//---------------------------------------------------------------------------------------------------------------
//
//  HAUD 2024.03.18
//
//  - XTS_TRANSPORT_LAYER
//
//  fb_TransportUnit
//  - Ctrl/STate interface, reacts to change of command
//    - Cmd(E_TRANSPORT_CTRL)
//
//  - controls members via structures and interfaces for getting XTS in defined state
//    - CMD_INIT:
//        - XPU is initialized:         XTS_CMD_INIT + PROGRESS_DONE
//        - XPU cyclic checks enabled:  XTS_IDLE     + PROGRESS_WORKING
//        - XPU detects mover:          _XpuState.Check == MOVER_ID_DETECTION_VALID
//
//    - CMD_IDLE
//      - Cyclic Checks of XPU and CaGroup
//        - XPU cyclic checks enabled:  XTS_IDLE     + PROGRESS_WORKING
//
//
//  CTRL / STATE --> see proprerties
//  structs for use of function block via mapping
//  cyclic check for new command
//
//  VAR INPUT / OUTPUT --> see properties
//
//---------------------------------------------------------------------------------------------------------------
// This SOFTWARE is provided as an Example by THE PROVIDER "as is" and "with all faults." THE PROVIDER makes no 
// representations or warranties of any kind concerning the safety, suitability, lack of viruses, inaccuracies, 
// typographical errors, or other harmful components of this SOFTWARE. There are inherent dangers in the use of 
// any software, and you are solely responsible for determining whether this SOFTWARE is compatible with your 
// equipment and other software installed on your equipment. You are also solely responsible for the protection 
// of your equipment and backup of your data, and THE PROVIDER will not be liable for any damages you may suffer 
// in connection with using, modifying, or distributing this SOFTWARE.
//---------------------------------------------------------------------------------------------------------------
FUNCTION_BLOCK fb_TransportUnit
VAR
  _eCheck                       : E_XTS_TRANSPORT_CHECK;

  // Transport Ctrl/State
  _stCtrl                       : REFERENCE TO ST_XTS_TRANSPORT_CTRL;
  _stState                      : REFERENCE TO ST_XTS_TRANSPORT_STATE;


  // execute transport commands
  _eCmd,
  _eCmdOld                      : E_XTS_TRANSPORT_CTRL;

  // execution state
  _eState                       : E_XTS_TRANSPORT_STATE;

  // execution result
  _eJobResult,
  _eResult                      : E_PROGRESS;


  // members of transport
  _XpuCtrl                      : REFERENCE TO ST_XPU_CTRL;                     // processing unit ctrl
  _XpuState                     : REFERENCE TO ST_XPU_STATE;                    // processing unit state
  _XpuInfo                      : REFERENCE TO ST_XPU_INFO;                     // processing unit information

  _GroupItf                     : I_XtsTransport_CaGroup;                       // group methods
  _GroupInfo                    : REFERENCE TO ST_GROUP_INFO;                   // info from group

  _MoverItf                     : REFERENCE TO ARRAY[1..MAX_MOVER] OF I_XtsTransport_Mover;   // mover methods
  _MoverInfo                    : REFERENCE TO ARRAY[1..MAX_MOVER] OF ST_MOVER_INFO;          // info from mover
  _MoverLastPosition            : REFERENCE TO ARRAY[1..MAX_MOVER] OF LREAL;                  // last commanded position of mover
  _MoverLastGap                 : REFERENCE TO ARRAY[1..MAX_MOVER] OF LREAL;                  // last commanded gapp of mover

  _StationStart                 : REFERENCE TO ST_STATION_PARAMETER;            // position, gap, dynamic constraints for sending all mover to start position

  // stations lists
  _ItfStationList               : REFERENCE TO ARRAY[1..MAX_STATION]  OF I_Station_LinkedList;  // access to all stations lists

  // station controls
  _StationControl               : REFERENCE TO ARRAY[1..MAX_STATION]  OF ST_STATION_CTRL;

  // station states
  _StationState                 : REFERENCE TO ARRAY[1..MAX_STATION]  OF ST_STATION_STATE;


  // access to stations methods by interface
  _ItfStationCtrl               : REFERENCE TO ARRAY[1..MAX_STATION]  OF I_XtsTransport_Station;

  _nStartStation                : UINT;

  _stMoverDataSend              : ST_STATION_MOVER_DATA;    // mover ticket data

  _stListResult                 : ST_STATION_LIST_RESULT;   // Xts station linkedlist entry

  _eMessageLevel                : E_MessageType;
  _stMsg                        : ST_Message;
END_VAR

IF NOT Check() THEN RETURN; END_IF

_stMsg.eDevice                  := XtsTransportUnit + 1;

_eCmd                           := _stCtrl.Cmd;
// check for command change
// get state for cmd
IF (_eCmd <> _eCmdOld)
THEN
  _eState                       := Cmd(_eCmd);
  _eCmdOld                      := _eCmd;

  IF (_eMessageLevel > E_MessageType.eMessageWarning)
  THEN
    _stMsg.eType                := E_MessageType.eMessageInfo;
    _stMsg.eSubdevice           := e_Subdevice.TransportUnit_General;
    _stMsg.iErrorNumber         := 0;
    _stMsg.sText                := concat( 'Command: ', TO_STRING(_eCmd));
    _stMsg.sText                := concat(_stMsg.sText, ': ');
    _stMsg.sText                := concat(_stMsg.sText, TO_STRING(_eResult));
    f_MessageSet(_stMsg);
  END_IF
END_IF

CASE _eResult
OF
  E_PROGRESS.PROGRESS_INVALID:
    _stState.State                := TO_UINT(_eResult);

  E_PROGRESS.PROGRESS_ERROR:
    _stState.State                := _eState + E_PROGRESS.PROGRESS_ERROR;

  E_PROGRESS.PROGRESS_DONE:
    _stState.State                := _eState + E_PROGRESS.PROGRESS_DONE;

    IF (_GroupInfo.GroupErrorStop) OR
       (_GroupInfo.GroupError)     OR
       NOT (_XpuInfo.AllPositionsValid)
    THEN
      _eResult                  := E_PROGRESS.PROGRESS_ERROR;
    END_IF
ELSE
  _stState.State                  := _eState + _eResult;

  CASE _eState
  OF
    E_XTS_TRANSPORT_STATE.TRANSPORT_INIT:
      _eResult                  := XpuInit(TRUE);
  
    E_XTS_TRANSPORT_STATE.TRANSPORT_IDLE:
      _eResult                  := f_GetProgress(_XpuState.State);
  
      IF (_GroupInfo.GroupErrorStop) OR
         (_GroupInfo.GroupError)     OR
         NOT (_XpuInfo.AllPositionsValid)
      THEN
        _eResult                := E_PROGRESS.PROGRESS_ERROR;
      END_IF
  
    E_XTS_TRANSPORT_STATE.TRANSPORT_MOVER_ENABLE:
      _eResult                  := MoverEnableAll(TRUE);
  
    E_XTS_TRANSPORT_STATE.TRANSPORT_MOVER_DISABLE:
      _eResult                  := MoverDisableAll(TRUE);

    E_XTS_TRANSPORT_STATE.TRANSPORT_MOVER_HALT_CA:
      _eResult                  := MoverHaltAll(TRUE);

    E_XTS_TRANSPORT_STATE.TRANSPORT_MOVER_STOP:
      _eResult                  := MoverStopAll(TRUE);
  
    E_XTS_TRANSPORT_STATE.TRANSPORT_GROUP_CLEAR:
      _eResult                  := GroupClear(TRUE);
  
    E_XTS_TRANSPORT_STATE.TRANSPORT_GROUP_BUILD:
      _eResult                  := GroupBuild(TRUE);
  
    E_XTS_TRANSPORT_STATE.TRANSPORT_GROUP_ENABLE:
      _eResult                  := GroupEnable(TRUE);

    E_XTS_TRANSPORT_STATE.TRANSPORT_GROUP_STOP:
      _eResult                  := GroupStop(TRUE);

    E_XTS_TRANSPORT_STATE.TRANSPORT_START:
      _eResult                  := TransportStart(TRUE);
  
    E_XTS_TRANSPORT_STATE.TRANSPORT_RESTART:
      _eResult                  := TransportRestart(TRUE);
  ELSE
    _eResult                    := E_PROGRESS.PROGRESS_INVALID;
  END_CASE

END_CASE

_stState.XpuState                 := _XpuState;
_stState.XpuInfo                  := _XpuInfo;
_stState.GroupInfo                := _GroupInfo;

METHOD PRIVATE Check  : BOOL
VAR_INST
  _idx        : UINT;
END_VAR

IF NOT __ISVALIDREF(_stCtrl)
THEN
  _eCheck                     := E_XTS_TRANSPORT_CHECK.POINTER_NULL_CTRL;
  RETURN;
END_IF

IF NOT __ISVALIDREF(_stState)
THEN
  _eCheck                     := E_XTS_TRANSPORT_CHECK.POINTER_NULL_STATE;
  RETURN;
END_IF

_stState.Check                  := _eCheck;

IF NOT __ISVALIDREF(_XpuCtrl)
THEN
  _eCheck                     := E_XTS_TRANSPORT_CHECK.POINTER_NULL_XPU_CTRL;
  RETURN;
END_IF

IF NOT __ISVALIDREF(_XpuState)
THEN
  _eCheck                     := E_XTS_TRANSPORT_CHECK.POINTER_NULL_XPU_STATE;
  RETURN;
END_IF

IF NOT __ISVALIDREF(_XpuInfo)
THEN
  _eCheck                     := E_XTS_TRANSPORT_CHECK.POINTER_NULL_XPU_INFO;
  RETURN;
END_IF

IF NOT (_GroupItf <> 0)
THEN
  _eCheck                     := E_XTS_TRANSPORT_CHECK.POINTER_NULL_GROUP_ITF;
  RETURN;
END_IF

IF NOT __ISVALIDREF(_GroupInfo)
THEN
  _eCheck                     := E_XTS_TRANSPORT_CHECK.POINTER_NULL_GROUP_INFO;
  RETURN;
END_IF

IF NOT __ISVALIDREF(_MoverItf)
THEN
  _eCheck                     := E_XTS_TRANSPORT_CHECK.POINTER_NULL_MOVER;
  RETURN;
END_IF

FOR _idx := 1 TO MAX_MOVER
DO
  IF NOT (_MoverItf[_idx] <> 0)
  THEN
    _eCheck                   := E_XTS_TRANSPORT_CHECK.POINTER_NULL_MOVER_ITF;
    RETURN;
  END_IF
END_FOR

IF NOT __ISVALIDREF(_MoverInfo)
THEN
  _eCheck                     := E_XTS_TRANSPORT_CHECK.POINTER_NULL_MOVER_INFO;
  RETURN;
END_IF

IF NOT __ISVALIDREF(_MoverLastPosition)
THEN
  _eCheck                     := E_XTS_TRANSPORT_CHECK.POINTER_NULL_MOVER_LAST_POS;
  RETURN;
END_IF

IF NOT __ISVALIDREF(_MoverLastGap)
THEN
  _eCheck                     := E_XTS_TRANSPORT_CHECK.POINTER_NULL_MOVER_LAST_GAP;
  RETURN;
END_IF

IF NOT __ISVALIDREF(_StationStart)
THEN
  _eCheck                     := E_XTS_TRANSPORT_CHECK.POINTER_NULL_STATION_START;
  RETURN;
END_IF

IF NOT __ISVALIDREF(_ItfStationList)
THEN
  _eCheck                     := E_XTS_TRANSPORT_CHECK.POINTER_NULL_STATION_ITF;
  RETURN;
END_IF

IF NOT __ISVALIDREF(_StationControl)
THEN
  _eCheck                     := E_XTS_TRANSPORT_CHECK.POINTER_NULL_STATION_CONTROL;
  RETURN;
END_IF

IF NOT __ISVALIDREF(_StationState)
THEN
  _eCheck                     := E_XTS_TRANSPORT_CHECK.POINTER_NULL_STATION_STATE;
  RETURN;
END_IF

IF NOT __ISVALIDREF(_ItfStationCtrl)
THEN
  _eCheck                     := E_XTS_TRANSPORT_CHECK.POINTER_NULL_STATION_CTRL_ITF;
  RETURN;
END_IF

FOR _idx := 1 TO MAX_STATION
DO
  IF NOT (_ItfStationCtrl[_idx] <> 0)
  THEN
    _eCheck                   := E_XTS_TRANSPORT_CHECK.POINTER_NULL_STATION_CTRL_ITF;
    RETURN;
  END_IF
END_FOR


_eCheck                       := E_XTS_TRANSPORT_CHECK.DONE_CHECK;
Check                         := TRUE;
END_METHOD

METHOD PRIVATE Cmd : E_XTS_TRANSPORT_STATE
VAR_INPUT
  Ctrl      : E_XTS_TRANSPORT_CTRL;
END_VAR
VAR_INST
  _eState   : E_XTS_TRANSPORT_STATE;
END_VAR
IF NOT Check() THEN RETURN; END_IF


CASE Ctrl
OF
  E_XTS_TRANSPORT_CTRL.CMD_NULL:  // clear all method calls
    _eState               := E_XTS_TRANSPORT_STATE.TRANSPORT_NULL;
    _eResult              := XpuInit         (FALSE);
    _eResult              := GroupClear      (FALSE);
    _eResult              := GroupBuild      (FALSE);
    _eResult              := GroupEnable     (FALSE);
    _eResult              := GroupStop       (FALSE);
    _eResult              := MoverEnableAll  (FALSE);
    _eResult              := MoverDisableAll (FALSE);
    _eResult              := MoverHaltAll    (FALSE);
    _eResult              := MoverStopAll    (FALSE);
    _eResult              := TransportStart  (FALSE);
    _eResult              := TransportRestart(FALSE);

  E_XTS_TRANSPORT_CTRL.CMD_INIT:  // clear methods for initialization
    _eState               := E_XTS_TRANSPORT_STATE.TRANSPORT_INIT;
    _eResult              := XpuInit(FALSE);


ELSE
  IF NOT (_XpuState.Init = E_XPU_INIT.INIT_DONE)
  THEN
    // no init, no further commands possible
    _eState               := E_XTS_TRANSPORT_STATE.TRANSPORT_INVALID;
  ELSE
    CASE Ctrl
    OF
      E_XTS_TRANSPORT_CTRL.CMD_IDLE:
        _eState           := E_XTS_TRANSPORT_STATE.TRANSPORT_IDLE;

      E_XTS_TRANSPORT_CTRL.CMD_MOVER_ENABLE:
        _eState           := E_XTS_TRANSPORT_STATE.TRANSPORT_MOVER_ENABLE;
        _eResult          := MoverEnableAll(FALSE);

      E_XTS_TRANSPORT_CTRL.CMD_MOVER_DISABLE:
        _eState           := E_XTS_TRANSPORT_STATE.TRANSPORT_MOVER_DISABLE;
        _eResult          := MoverDisableAll(FALSE);

      E_XTS_TRANSPORT_CTRL.CMD_MOVER_HALT_CA:
        _eState           := E_XTS_TRANSPORT_STATE.TRANSPORT_MOVER_HALT_CA;
        _eResult          := MoverHaltAll(FALSE);

      E_XTS_TRANSPORT_CTRL.CMD_MOVER_STOP:
        _eState           := E_XTS_TRANSPORT_STATE.TRANSPORT_MOVER_STOP;
        _eResult          := MoverStopAll(FALSE);

      E_XTS_TRANSPORT_CTRL.CMD_GROUP_CLEAR:
        _eState           := E_XTS_TRANSPORT_STATE.TRANSPORT_GROUP_CLEAR;
        _eResult          := GroupClear (FALSE);

      E_XTS_TRANSPORT_CTRL.CMD_GROUP_BUILD:
        _eState           := E_XTS_TRANSPORT_STATE.TRANSPORT_GROUP_BUILD;
        _eResult          := GroupBuild (FALSE);

      E_XTS_TRANSPORT_CTRL.CMD_GROUP_ENABLE:
        _eState           := E_XTS_TRANSPORT_STATE.TRANSPORT_GROUP_ENABLE;
        _eResult          := GroupEnable(FALSE);

      E_XTS_TRANSPORT_CTRL.CMD_GROUP_STOP:
        _eState           := E_XTS_TRANSPORT_STATE.TRANSPORT_GROUP_STOP;
        _eResult          := GroupStop(FALSE);

      E_XTS_TRANSPORT_CTRL.CMD_TRANSPORT_START:
        _eState           := E_XTS_TRANSPORT_STATE.TRANSPORT_START;
        _eResult          := TransportStart(FALSE);

      E_XTS_TRANSPORT_CTRL.CMD_TRANSPORT_RESTART:
        _eState           := E_XTS_TRANSPORT_STATE.TRANSPORT_RESTART;
        _eResult          := TransportRestart(FALSE);

    ELSE
        _eState           := E_XTS_TRANSPORT_STATE.TRANSPORT_INVALID;
    END_CASE
  END_IF
END_CASE

Cmd                       := _eState;
END_METHOD

PROPERTY Ctrl : REFERENCE TO ST_XTS_TRANSPORT_CTRL
SET
_stCtrl REF= Ctrl;
END_SET
END_PROPERTY

METHOD GroupBuild : E_PROGRESS
VAR_INPUT
  Execute     : BOOL;
END_VAR
VAR_INST
  _nErrorId   : UDINT;
  _eJobReslt,
  _eState     : E_PROGRESS;
END_VAR
//-----------------------------------------------------------------------------
IF NOT Execute 
THEN 
	_eState                       := E_PROGRESS.PROGRESS_INIT; 
END_IF 
//-----------------------------------------------------------------------------
IF NOT Check() 
THEN 
	GroupBuild                    := E_PROGRESS.PROGRESS_ERROR; 
	RETURN; 
END_IF
//-----------------------------------------------------------------------------
//-----------------------------------------------------------------------------
CASE _eState
OF
  E_PROGRESS.PROGRESS_INIT:
    IF Execute
    THEN
      _nErrorId                 := 0;

      IF (_GroupInfo.AxisCount <> 0)
      THEN
        _nErrorId               := 9999;
        _eState                 := E_PROGRESS.PROGRESS_ERROR;

        _stMsg.eType            := E_MessageType.eMessageError;
        _stMsg.eSubdevice       := e_Subdevice.TransportUnit_GroupBuild;
        _stMsg.iErrorNumber     := _nErrorId;
        _stMsg.sText            := concat( 'State: ', TO_STRING(THIS^._eState));
        _stMsg.sText            := concat(_stMsg.sText, ': ');
        _stMsg.sText            := concat(_stMsg.sText, TO_STRING(_eState));
        f_MessageSet(_stMsg);
      ELSE
        _eState                 := E_PROGRESS.PROGRESS_BUSY;
        _eJobReslt              := _GroupItf.AddAll(FALSE);

        IF (_eMessageLevel > E_MessageType.eMessageError)
        THEN
          _stMsg.eType          := E_MessageType.eMessageinfo;
          _stMsg.eSubdevice     := e_Subdevice.TransportUnit_GroupBuild;
          _stMsg.iErrorNumber   := 0;
          _stMsg.sText          := concat( 'State: ', TO_STRING(THIS^._eState));
          _stMsg.sText          := concat(_stMsg.sText, ': ');
          _stMsg.sText          := concat(_stMsg.sText, TO_STRING(_eState));
          f_MessageSet(_stMsg);
        END_IF
      END_IF
    END_IF
END_CASE
//---------------------------------------------------------------------------
//---------------------------------------------------------------------------
CASE _eState
OF
  E_PROGRESS.PROGRESS_BUSY:
    _eJobReslt                  := _GroupItf.AddAll(TRUE);

    IF (_eJobReslt = E_PROGRESS.PROGRESS_ERROR)
    THEN
      _eState                   := E_PROGRESS.PROGRESS_ERROR;

      _nErrorId                 := _GroupInfo.GroupErrorId;
      _eJobReslt                := _GroupItf.AddAll(FALSE);

    ELSIF (_eJobReslt = E_PROGRESS.PROGRESS_DONE)
    THEN
      _eState                   := E_PROGRESS.PROGRESS_PREPARE;
      _eJobReslt                := _GroupItf.AddAll(FALSE);
	    _eJobReslt				        := _GroupItf.Reset(FALSE);
    END_IF
END_CASE
//-----------------------------------------------------------------------------
//-----------------------------------------------------------------------------
CASE _eState
OF
  E_PROGRESS.PROGRESS_PREPARE:
    _eJobReslt                  := _GroupItf.Reset(TRUE);

    IF (_eJobReslt = E_PROGRESS.PROGRESS_ERROR)
    THEN
      _eState                   := E_PROGRESS.PROGRESS_ERROR;

      _nErrorId                 := _GroupInfo.GroupErrorId;
	    _eJobReslt				        := _GroupItf.Reset(FALSE);

    ELSIF (_eJobReslt = E_PROGRESS.PROGRESS_DONE)
    THEN
      _eState                   := E_PROGRESS.PROGRESS_DONE;
	    _eJobReslt				        := _GroupItf.Reset(FALSE);

      IF (_eMessageLevel > E_MessageType.eMessageError)
      THEN
        _stMsg.eType            := E_MessageType.eMessageInfo;
        _stMsg.eSubdevice       := e_Subdevice.TransportUnit_General;
        _stMsg.iErrorNumber     := 0;
        _stMsg.sText            := concat( 'State: ', TO_STRING(THIS^._eState));
        _stMsg.sText            := concat(_stMsg.sText, ': ');
        _stMsg.sText            := concat(_stMsg.sText, TO_STRING(_eState));
        f_MessageSet(_stMsg);
      END_IF
    END_IF
END_CASE
//-----------------------------------------------------------------------------
//-----------------------------------------------------------------------------

GroupBuild                      := _eState;
END_METHOD

METHOD GroupClear : E_PROGRESS
VAR_INPUT
  Execute     : BOOL;
END_VAR
VAR_INST
  _nRepeat,
  _nStation,
  _nErrorId   : UDINT;
  _eJobReslt,
  _eState     : E_PROGRESS;
END_VAR
//-----------------------------------------------------------------------------
IF NOT Execute 
THEN 
	_eState                       := E_PROGRESS.PROGRESS_INIT; 
END_IF 
//-----------------------------------------------------------------------------
IF NOT Check() 
THEN 
	GroupClear                    := E_PROGRESS.PROGRESS_ERROR; 
	RETURN; 
END_IF
//-----------------------------------------------------------------------------
//-----------------------------------------------------------------------------
CASE _eState
OF
  E_PROGRESS.PROGRESS_INIT:
    IF Execute
    THEN
      _nRepeat                  :=
      _nErrorId                 := 0;
      _eJobReslt                := _GroupItf.McHaltAll(FALSE);
      _eJobReslt                := _GroupItf.RemoveAll(FALSE);
      _eJobReslt                := _GroupItf.McResetAll(FALSE);
      _eJobReslt                := _GroupItf.Disable(FALSE);
      _eJobReslt                := _GroupItf.Reset(FALSE);
      _eJobReslt                := StationsClearOutfeed(FALSE);

      _eState                   := E_PROGRESS.PROGRESS_BUSY;

      IF (_eMessageLevel > E_MessageType.eMessageError)
      THEN
        _stMsg.eType            := E_MessageType.eMessageinfo;
        _stMsg.eSubdevice       := e_Subdevice.TransportUnit_GroupClear;
        _stMsg.iErrorNumber     := 0;
        _stMsg.sText            := concat( 'State: ', TO_STRING(THIS^._eState));
        _stMsg.sText            := concat(_stMsg.sText, ': ');
        _stMsg.sText            := concat(_stMsg.sText, TO_STRING(_eState));
        f_MessageSet(_stMsg);
      END_IF
    END_IF
END_CASE
//---------------------------------------------------------------------------
//---------------------------------------------------------------------------
CASE _eState
OF
  E_PROGRESS.PROGRESS_BUSY:
    _eJobReslt                  := StationsClearOutfeed(TRUE);

    IF (_eJobReslt = E_PROGRESS.PROGRESS_DONE)
    THEN
      _eState                   := E_PROGRESS.PROGRESS_PREPARE;
      _eJobReslt                := StationsClearOutfeed(FALSE);
    END_IF

  //---------------------------------------------------------------------------
  //---------------------------------------------------------------------------
  E_PROGRESS.PROGRESS_PREPARE:
    _eJobReslt                  := _GroupItf.McHaltAll(TRUE);

    IF (_eJobReslt > E_PROGRESS.PROGRESS_STILL_WORKING)
    THEN
      _eState                   := E_PROGRESS.PROGRESS_STARTUP;
      _nErrorId                 := _GroupInfo.GroupErrorId;
      _eJobReslt                := _GroupItf.McHaltAll(FALSE);
    END_IF
  //---------------------------------------------------------------------------
  //---------------------------------------------------------------------------
  E_PROGRESS.PROGRESS_STARTUP:
    _eJobReslt                  := _GroupItf.RemoveAll(TRUE);

    IF (_eJobReslt > E_PROGRESS.PROGRESS_STILL_WORKING)
    THEN
      _eState                   := E_PROGRESS.PROGRESS_CHECK;
      _nErrorId                 := _GroupInfo.GroupErrorId;
      _eJobReslt                := _GroupItf.RemoveAll(FALSE);
    END_IF
  //---------------------------------------------------------------------------
  //---------------------------------------------------------------------------
  E_PROGRESS.PROGRESS_CHECK:
    _eJobReslt                  := _GroupItf.Disable(TRUE);

    IF (_eJobReslt > E_PROGRESS.PROGRESS_STILL_WORKING)
    THEN
      _eState                   := E_PROGRESS.PROGRESS_OCCUPIED;
      _nErrorId                 := _GroupInfo.GroupErrorId;
      _eJobReslt                := _GroupItf.Disable(FALSE);
    END_IF
  //---------------------------------------------------------------------------
  //---------------------------------------------------------------------------
  E_PROGRESS.PROGRESS_OCCUPIED:
    _eJobReslt                  := _GroupItf.Reset(TRUE);

    IF (_eJobReslt > E_PROGRESS.PROGRESS_STILL_WORKING)
    THEN
      _eState                   := E_PROGRESS.PROGRESS_WORKING;
      _nErrorId                 := _GroupInfo.GroupErrorId;
      _eJobReslt                := _GroupItf.Reset(FALSE);
    END_IF
END_CASE
//-----------------------------------------------------------------------------
//-----------------------------------------------------------------------------
CASE _eState
OF
  E_PROGRESS.PROGRESS_WORKING:
    IF    (_GroupInfo.AxisCount     = 0) AND
          (_GroupInfo.CaGroupState  = E_CA_GROUP_STATE.mcGroupStateDisabled) AND 
      NOT (_GroupInfo.GroupError)
    THEN
      _eState                   := E_PROGRESS.PROGRESS_DONE;

      IF (_eMessageLevel > E_MessageType.eMessageError)
      THEN
        _stMsg.eType            := E_MessageType.eMessageInfo;
        _stMsg.eSubdevice       := e_Subdevice.TransportUnit_GroupClear;
        _stMsg.iErrorNumber     := 0;
        _stMsg.sText            := concat( 'State: ', TO_STRING(THIS^._eState));
        _stMsg.sText            := concat(_stMsg.sText, ': ');
        _stMsg.sText            := concat(_stMsg.sText, TO_STRING(_eState));
        f_MessageSet(_stMsg);
      END_IF
      GVL_MSG_XTS.TransportMessageCtrl.Cmd  := E_MESSAGE_CTRL.MSG_CTRL_WRITE;
    ELSE
      _nRepeat                  := _nRepeat + 1;
      IF NOT (_nRepeat > 2)
      THEN
        _eState                 := E_PROGRESS.PROGRESS_BUSY;
      ELSE
        _eState                 := E_PROGRESS.PROGRESS_ERROR;
      END_IF
    END_IF
END_CASE
//-----------------------------------------------------------------------------
//-----------------------------------------------------------------------------

GroupClear                      := _eState;
END_METHOD

METHOD GroupEnable : E_PROGRESS
VAR_INPUT
  Execute     : BOOL;
END_VAR
VAR_INST
  _nErrorId   : UDINT;
  _eJobReslt,
  _eState     : E_PROGRESS;
END_VAR
//-----------------------------------------------------------------------------
IF NOT Execute 
THEN 
	_eState                       := E_PROGRESS.PROGRESS_INIT; 
END_IF 
//-----------------------------------------------------------------------------
IF NOT Check() 
THEN 
	GroupEnable                   := E_PROGRESS.PROGRESS_ERROR; 
	RETURN; 
END_IF
//-----------------------------------------------------------------------------
//-----------------------------------------------------------------------------
CASE _eState
OF
  E_PROGRESS.PROGRESS_INIT:
    IF Execute
    THEN
      _nErrorId                 := 0;

      IF NOT (_GroupInfo.AxisCount <> 0)
      THEN
        _nErrorId               := 9999;
        _eState                 := E_PROGRESS.PROGRESS_ERROR;

        _stMsg.eType            := E_MessageType.eMessageError;
        _stMsg.eSubdevice       := e_Subdevice.TransportUnit_GroupEnable;
        _stMsg.iErrorNumber     := _nErrorId;
        _stMsg.sText            := concat( 'State: ', TO_STRING(THIS^._eState));
        _stMsg.sText            := concat(_stMsg.sText, ': ');
        _stMsg.sText            := concat(_stMsg.sText, TO_STRING(_eState));
        f_MessageSet(_stMsg);
      ELSE
        _eState                 := E_PROGRESS.PROGRESS_BUSY;
        _eJobReslt              := _GroupItf.Enable(FALSE);

        IF (_eMessageLevel > E_MessageType.eMessageError)
        THEN
          _stMsg.eType          := E_MessageType.eMessageinfo;
          _stMsg.eSubdevice     := e_Subdevice.TransportUnit_GroupEnable;
          _stMsg.iErrorNumber   := 0;
          _stMsg.sText          := concat( 'State: ', TO_STRING(THIS^._eState));
          _stMsg.sText          := concat(_stMsg.sText, ': ');
          _stMsg.sText          := concat(_stMsg.sText, TO_STRING(_eState));
          f_MessageSet(_stMsg);
        END_IF

      END_IF
    END_IF
END_CASE
//---------------------------------------------------------------------------
//---------------------------------------------------------------------------
CASE _eState
OF
  E_PROGRESS.PROGRESS_BUSY:
    _eJobReslt                  := _GroupItf.Enable(TRUE);

    IF (_eJobReslt = E_PROGRESS.PROGRESS_ERROR)
    THEN
      _eState                   := E_PROGRESS.PROGRESS_ERROR;

      _nErrorId                 := _GroupInfo.GroupErrorId;
      _eJobReslt                := _GroupItf.Enable(FALSE);

    ELSIF (_eJobReslt = E_PROGRESS.PROGRESS_DONE)
    THEN
      _eState                   := E_PROGRESS.PROGRESS_CHECK;
      _eJobReslt                := _GroupItf.Enable(FALSE);
    END_IF
END_CASE
//-----------------------------------------------------------------------------
//-----------------------------------------------------------------------------
CASE _eState
OF
  E_PROGRESS.PROGRESS_CHECK:
    IF (_GroupInfo.GroupStandby) OR
       (_GroupInfo.GroupMoving)  OR
       (_GroupInfo.GroupNotReady)
    THEN
      _eState                   := E_PROGRESS.PROGRESS_DONE;

      IF (_eMessageLevel > E_MessageType.eMessageError)
      THEN
        _stMsg.eType            := E_MessageType.eMessageinfo;
        _stMsg.eSubdevice       := e_Subdevice.TransportUnit_GroupEnable;
        _stMsg.iErrorNumber     := 0;
        _stMsg.sText            := concat( 'State: ', TO_STRING(THIS^._eState));
        _stMsg.sText            := concat(_stMsg.sText, ': ');
        _stMsg.sText            := concat(_stMsg.sText, TO_STRING(_eState));
        f_MessageSet(_stMsg);
      END_IF
    ELSE
      IF (_GroupInfo.GroupErrorStop) OR
         (_GroupInfo.GroupError)
      THEN
        _eState                 := E_PROGRESS.PROGRESS_ERROR;
      END_IF
    END_IF
END_CASE
//-----------------------------------------------------------------------------
//-----------------------------------------------------------------------------
GroupEnable                     := _eState;
END_METHOD

PROPERTY GroupInfo : REFERENCE TO ST_GROUP_INFO
SET
_GroupInfo REF= GroupInfo;
END_SET
END_PROPERTY

PROPERTY GroupItf : I_XtsTransport_CaGroup
SET
_GroupItf := GroupItf;
END_SET
END_PROPERTY

METHOD GroupStop : E_PROGRESS
VAR_INPUT
  Execute     : BOOL;
END_VAR
VAR_INST
  _nRepeat,
  _nStation,
  _nErrorId   : UDINT;
  _eJobReslt,
  _eState     : E_PROGRESS;
END_VAR
//-----------------------------------------------------------------------------
IF NOT Execute 
THEN 
	_eState                      := E_PROGRESS.PROGRESS_INIT; 
END_IF 
//-----------------------------------------------------------------------------
IF NOT Check() 
THEN 
	GroupStop                    := E_PROGRESS.PROGRESS_ERROR; 
	RETURN; 
END_IF
//-----------------------------------------------------------------------------
//-----------------------------------------------------------------------------
CASE _eState
OF
  E_PROGRESS.PROGRESS_INIT:
    IF Execute
    THEN
      _nRepeat                  :=
      _nErrorId                 := 0;
      _eJobReslt                := _GroupItf.Stop(FALSE);

      _eState                   := E_PROGRESS.PROGRESS_BUSY;

      IF (_eMessageLevel > E_MessageType.eMessageError)
      THEN
        _stMsg.eType            := E_MessageType.eMessageinfo;
        _stMsg.eSubdevice       := e_Subdevice.TransportUnit_GroupStop;
        _stMsg.iErrorNumber     := 0;
        _stMsg.sText            := concat( 'State: ', TO_STRING(THIS^._eState));
        _stMsg.sText            := concat(_stMsg.sText, ': ');
        _stMsg.sText            := concat(_stMsg.sText, TO_STRING(_eState));
        f_MessageSet(_stMsg);
      END_IF
    END_IF
END_CASE
//---------------------------------------------------------------------------
//---------------------------------------------------------------------------
CASE _eState
OF
  E_PROGRESS.PROGRESS_BUSY:
    _eJobReslt                  := _GroupItf.Stop(TRUE);

    IF (_eJobReslt = E_PROGRESS.PROGRESS_ERROR)
    THEN
      _eState                   := E_PROGRESS.PROGRESS_PREPARE;
      _nErrorId                 := _GroupInfo.GroupErrorId;
      _eJobReslt                := _GroupItf.Stop(FALSE);

    ELSIF (_eJobReslt = E_PROGRESS.PROGRESS_DONE)
    THEN
      _eState                   := E_PROGRESS.PROGRESS_WORKING;
      _eJobReslt                := _GroupItf.Stop(FALSE);
    END_IF
END_CASE
//-----------------------------------------------------------------------------
//-----------------------------------------------------------------------------
CASE _eState
OF
  E_PROGRESS.PROGRESS_WORKING:
    IF NOT (_GroupInfo.GroupError)
    THEN
      _eState                   := E_PROGRESS.PROGRESS_DONE;

      IF (_eMessageLevel > E_MessageType.eMessageError)
      THEN
        _stMsg.eType            := E_MessageType.eMessageInfo;
        _stMsg.eSubdevice       := e_Subdevice.TransportUnit_General;
        _stMsg.iErrorNumber     := 0;
        _stMsg.sText            := concat( 'State: ', TO_STRING(THIS^._eState));
        _stMsg.sText            := concat(_stMsg.sText, ': ');
        _stMsg.sText            := concat(_stMsg.sText, TO_STRING(_eState));
        f_MessageSet(_stMsg);
      END_IF
    ELSE
      IF (_GroupInfo.GroupErrorStop) OR
         (_GroupInfo.GroupError)
      THEN
        _nRepeat                := _nRepeat + 1;
        IF NOT (_nRepeat > 2)
        THEN
          _eState               := E_PROGRESS.PROGRESS_BUSY;
        ELSE
          _eState               := E_PROGRESS.PROGRESS_ERROR;
        END_IF
      END_IF
    END_IF
END_CASE
//-----------------------------------------------------------------------------
//-----------------------------------------------------------------------------

GroupStop                       := _eState;
END_METHOD

PROPERTY MessageLevel : e_messagetype
SET
_eMessageLevel := MessageLevel;
END_SET
END_PROPERTY

METHOD MoverDisableAll : e_progress
VAR_INPUT
  Execute     : BOOL;
END_VAR
VAR_INST
  _nMover     : UINT;
  _nErrorId   : UDINT;
  _eRslt,
  _eState     : E_PROGRESS;
END_VAR
//-----------------------------------------------------------------------------
IF NOT Execute 
THEN 
	_eState                       := E_PROGRESS.PROGRESS_INIT; 
END_IF 
//-----------------------------------------------------------------------------
IF NOT Check() 
THEN 
	MoverDisableAll               := E_PROGRESS.PROGRESS_ERROR; 
	RETURN; 
END_IF
//-----------------------------------------------------------------------------
//-----------------------------------------------------------------------------
CASE _eState
OF
  E_PROGRESS.PROGRESS_INIT:
    IF Execute
    THEN
      _nErrorId                 := 0;
      _nMover                   := 1;

      _eState                   := E_PROGRESS.PROGRESS_BUSY;

      IF (_eMessageLevel > E_MessageType.eMessageError)
      THEN
        _stMsg.eType            := E_MessageType.eMessageinfo;
        _stMsg.eSubdevice       := e_Subdevice.TransportUnit_MoverDisableAll;
        _stMsg.iErrorNumber     := 0;
        _stMsg.sText            := concat( 'State: ', TO_STRING(THIS^._eState));
        _stMsg.sText            := concat(_stMsg.sText, ': ');
        _stMsg.sText            := concat(_stMsg.sText, TO_STRING(_eState));
        f_MessageSet(_stMsg);
      END_IF
    END_IF
END_CASE
//-----------------------------------------------------------------------------
//-----------------------------------------------------------------------------
CASE _eState
OF
  E_PROGRESS.PROGRESS_BUSY:
    _eState                     := E_PROGRESS.PROGRESS_PREPARE;
    _eRslt                      := _MoverItf[_nMover].Disable(FALSE);
    _eRslt                      := _MoverItf[_nMover].Reset(FALSE);
END_CASE
//-----------------------------------------------------------------------------
//-----------------------------------------------------------------------------
CASE _eState
OF
  E_PROGRESS.PROGRESS_PREPARE:
    _eRslt                      := _MoverItf[_nMover].Disable(TRUE);

    IF (_eRslt = E_PROGRESS.PROGRESS_ERROR)
    THEN
      _eState                   := E_PROGRESS.PROGRESS_BUSY;
      _nErrorId                 := _MoverInfo[_nMover].nErrorId; 
      _eRslt                    := _MoverItf[_nMover].Disable(FALSE);
      _MoverItf[_nMover].Reset(TRUE);

    ELSIF (_eRslt = E_PROGRESS.PROGRESS_DONE)
    THEN
      _eState                   := E_PROGRESS.PROGRESS_STARTUP;
    END_IF
END_CASE
//-----------------------------------------------------------------------------
//-----------------------------------------------------------------------------
CASE _eState
OF
  E_PROGRESS.PROGRESS_STARTUP:
    _eState                     := E_PROGRESS.PROGRESS_CHECK;
    _eRslt                      := _MoverItf[_nMover].Disable(FALSE);
END_CASE
//-----------------------------------------------------------------------------
//-----------------------------------------------------------------------------
CASE _eState
OF
  E_PROGRESS.PROGRESS_CHECK:
    IF (_nMover > GVL_XTS.XpuInfo.nDetectedAxisCount-1)
    THEN
      _eState                   := E_PROGRESS.PROGRESS_DONE;

      IF (_eMessageLevel > E_MessageType.eMessageError)
      THEN
        _stMsg.eType            := E_MessageType.eMessageInfo;
        _stMsg.eSubdevice       := e_Subdevice.TransportUnit_General;
        _stMsg.iErrorNumber     := 0;
        _stMsg.sText            := concat( 'State: ', TO_STRING(THIS^._eState));
        _stMsg.sText            := concat(_stMsg.sText, ': ');
        _stMsg.sText            := concat(_stMsg.sText, TO_STRING(_eState));
        f_MessageSet(_stMsg);
      END_IF
    ELSE
      _nMover                   := _nMover + 1;
      _eState                   := E_PROGRESS.PROGRESS_BUSY;
    END_IF
END_CASE
//-----------------------------------------------------------------------------
//-----------------------------------------------------------------------------

MoverDisableAll                 := _eState;
END_METHOD

METHOD MoverEnableAll : e_progress
VAR_INPUT
  Execute     : BOOL;
END_VAR
VAR_INST
  _nMover     : UINT;
  _nErrorId   : UDINT;
  _eRslt,
  _eState     : E_PROGRESS;
END_VAR
//-----------------------------------------------------------------------------
IF NOT Execute 
THEN 
	_eState                       := E_PROGRESS.PROGRESS_INIT; 
END_IF 
//-----------------------------------------------------------------------------
IF NOT Check() 
THEN 
	MoverEnableAll                := E_PROGRESS.PROGRESS_ERROR; 
	RETURN; 
END_IF
//-----------------------------------------------------------------------------
//-----------------------------------------------------------------------------
CASE _eState
OF
  E_PROGRESS.PROGRESS_INIT:
    IF Execute
    THEN
      _nErrorId                 := 0;
      _nMover                   := 1;

      _eState                   := E_PROGRESS.PROGRESS_BUSY;

      IF (_eMessageLevel > E_MessageType.eMessageError)
      THEN
        _stMsg.eType            := E_MessageType.eMessageinfo;
        _stMsg.eSubdevice       := e_Subdevice.TransportUnit_MoverEnableAll;
        _stMsg.iErrorNumber     := 0;
        _stMsg.sText            := concat( 'State: ', TO_STRING(THIS^._eState));
        _stMsg.sText            := concat(_stMsg.sText, ': ');
        _stMsg.sText            := concat(_stMsg.sText, TO_STRING(_eState));
        f_MessageSet(_stMsg);
      END_IF
    END_IF
END_CASE
//-----------------------------------------------------------------------------
//-----------------------------------------------------------------------------
CASE _eState
OF
  E_PROGRESS.PROGRESS_BUSY:
    _eState                     := E_PROGRESS.PROGRESS_PREPARE;
    _eRslt                      := _MoverItf[_nMover].Enable(FALSE);
    _eRslt                      := _MoverItf[_nMover].Reset (FALSE);
END_CASE
//-----------------------------------------------------------------------------
//-----------------------------------------------------------------------------
CASE _eState
OF
  E_PROGRESS.PROGRESS_PREPARE:
    _eRslt                      := _MoverItf[_nMover].Enable(TRUE);

    IF (_eRslt = E_PROGRESS.PROGRESS_ERROR)
    THEN
      _eState                   := E_PROGRESS.PROGRESS_BUSY;
      _nErrorId                 := _MoverInfo[_nMover].nErrorId;
      _MoverItf[_nMover].Reset (TRUE);

    ELSIF (_eRslt = E_PROGRESS.PROGRESS_DONE)
    THEN
      _eState                   := E_PROGRESS.PROGRESS_STARTUP;
    END_IF
END_CASE
//-----------------------------------------------------------------------------
//-----------------------------------------------------------------------------
CASE _eState
OF
  E_PROGRESS.PROGRESS_STARTUP:
    _eState                     := E_PROGRESS.PROGRESS_CHECK;
    _eRslt                      := _MoverItf[_nMover].Enable(FALSE);
END_CASE
//-----------------------------------------------------------------------------
//-----------------------------------------------------------------------------
CASE _eState
OF
  E_PROGRESS.PROGRESS_CHECK:
    IF (_nMover > GVL_XTS.XpuInfo.nDetectedAxisCount-1)
    THEN
      _eState                   := E_PROGRESS.PROGRESS_DONE;
      IF (_eMessageLevel > E_MessageType.eMessageError)
      THEN
        _stMsg.eType            := E_MessageType.eMessageInfo;
        _stMsg.eSubdevice       := e_Subdevice.TransportUnit_General;
        _stMsg.iErrorNumber     := 0;
        _stMsg.sText            := concat( 'State: ', TO_STRING(THIS^._eState));
        _stMsg.sText            := concat(_stMsg.sText, ': ');
        _stMsg.sText            := concat(_stMsg.sText, TO_STRING(_eState));
        f_MessageSet(_stMsg);
      END_IF
    ELSE
      _nMover                   := _nMover + 1;
      _eState                   := E_PROGRESS.PROGRESS_BUSY;
    END_IF
END_CASE
//-----------------------------------------------------------------------------
//-----------------------------------------------------------------------------

MoverEnableAll                  := _eState;
END_METHOD

METHOD MoverHaltAll : e_progress
VAR_INPUT
  Execute     : BOOL;
END_VAR
VAR_INST
  _nMover     : UINT;
  _nErrorId   : UDINT;
  _eRslt,
  _eState     : E_PROGRESS;
  _stMoveData : ST_MOVE_DATA; // dyn constraints for _MoverItf[i].Halt(Execute, stMoveData)
END_VAR
//-----------------------------------------------------------------------------
IF NOT Execute 
THEN 
	_eState                       := E_PROGRESS.PROGRESS_INIT; 
END_IF 
//-----------------------------------------------------------------------------
IF NOT Check() 
THEN 
	MoverHaltAll                  := E_PROGRESS.PROGRESS_ERROR; 
	RETURN; 
END_IF
//-----------------------------------------------------------------------------
//-----------------------------------------------------------------------------
CASE _eState
OF
  E_PROGRESS.PROGRESS_INIT:
    IF Execute
    THEN
      _nErrorId                 := 0;
      _nMover                   := 1;

      _eState                   := E_PROGRESS.PROGRESS_BUSY;

      IF (_eMessageLevel > E_MessageType.eMessageError)
      THEN
        _stMsg.eType            := E_MessageType.eMessageinfo;
        _stMsg.iErrorNumber     := 0;
        _stMsg.sText            := concat( 'State: ', TO_STRING(THIS^._eState));
        _stMsg.sText            := concat(_stMsg.sText, ': ');
        _stMsg.sText            := concat(_stMsg.sText, TO_STRING(_eState));
        f_MessageSet(_stMsg);
      END_IF
    END_IF
END_CASE
//-----------------------------------------------------------------------------
//-----------------------------------------------------------------------------
CASE _eState
OF
  E_PROGRESS.PROGRESS_BUSY:
    _eState                     := E_PROGRESS.PROGRESS_PREPARE;
    _stMoveData.rAcc            := _StationStart.rAccDec;
    _stMoveData.rGap            := _MoverLastGap[_nMover];

    IF NOT (_GroupInfo.AxisCount = GVL_XTS.XpuInfo.nDetectedAxisCount)
    THEN
      _eRslt                    := _MoverItf[_nMover].Halt(FALSE, _stMoveData);
    ELSE
      _eRslt                    := _MoverItf[_nMover].HaltCa(FALSE, _stMoveData);
    END_IF
END_CASE
//-----------------------------------------------------------------------------
//-----------------------------------------------------------------------------
CASE _eState
OF
  E_PROGRESS.PROGRESS_PREPARE:
    IF NOT (_GroupInfo.AxisCount = GVL_XTS.XpuInfo.nDetectedAxisCount)
    THEN
      _eRslt                    := _MoverItf[_nMover].Halt(TRUE, _stMoveData);
    ELSE
      _eRslt                    := _MoverItf[_nMover].HaltCa(TRUE, _stMoveData);
    END_IF

    IF (_eRslt = E_PROGRESS.PROGRESS_ERROR)
    THEN
      _eState                   := E_PROGRESS.PROGRESS_WORKING; // reset error on purpose, since we have to come back and get everybody in standstill
      _eRslt                    := _MoverItf[_nMover].Reset(FALSE);
      _nErrorId                 := _MoverInfo[_nMover].nErrorId; 

    ELSIF (_eRslt = E_PROGRESS.PROGRESS_DONE)
    THEN
      _eState                   := E_PROGRESS.PROGRESS_STARTUP;
    END_IF
END_CASE
//-----------------------------------------------------------------------------
//-----------------------------------------------------------------------------
CASE _eState
OF
  E_PROGRESS.PROGRESS_STARTUP:
    _eState                     := E_PROGRESS.PROGRESS_CHECK;

    IF NOT (_GroupInfo.AxisCount = MAX_MOVER)
    THEN
      _eRslt                    := _MoverItf[_nMover].Halt(FALSE, _stMoveData);
    ELSE
      _eRslt                    := _MoverItf[_nMover].HaltCa(FALSE, _stMoveData);
    END_IF

END_CASE
//-----------------------------------------------------------------------------
//-----------------------------------------------------------------------------
CASE _eState
OF
  E_PROGRESS.PROGRESS_CHECK:
    IF (_nMover > GVL_XTS.XpuInfo.nDetectedAxisCount-1)
    THEN
      _eState                   := E_PROGRESS.PROGRESS_OCCUPIED;
    ELSE
      _nMover                   := _nMover + 1;
      _eState                   := E_PROGRESS.PROGRESS_BUSY;
    END_IF
END_CASE
//-----------------------------------------------------------------------------
//-----------------------------------------------------------------------------
CASE _eState
OF
  E_PROGRESS.PROGRESS_OCCUPIED:
    IF (_GroupInfo.AllAxesStanding)
    THEN
      _eState                   := E_PROGRESS.PROGRESS_DONE;

      IF (_eMessageLevel > E_MessageType.eMessageError)
      THEN
        _stMsg.eType            := E_MessageType.eMessageInfo;
        _stMsg.eSubdevice       := e_Subdevice.TransportUnit_General;
        _stMsg.iErrorNumber     := 0;
        _stMsg.sText            := concat( 'State: ', TO_STRING(THIS^._eState));
        _stMsg.sText            := concat(_stMsg.sText, ': ');
        _stMsg.sText            := concat(_stMsg.sText, TO_STRING(_eState));
        f_MessageSet(_stMsg);
      END_IF
    ELSE
      _nMover                   := 1;
      _eState                   := E_PROGRESS.PROGRESS_BUSY;
    END_IF
END_CASE
//-----------------------------------------------------------------------------
//-----------------------------------------------------------------------------
CASE _eState
OF
  E_PROGRESS.PROGRESS_WORKING:
    _eRslt                      := _MoverItf[_nMover].Reset(TRUE);

    IF (_eRslt = E_PROGRESS.PROGRESS_ERROR)
    THEN
      _eRslt                    := _MoverItf[_nMover].Reset(FALSE);
      _nErrorId                 := _MoverInfo[_nMover].nErrorId; 

    ELSIF (_eRslt = E_PROGRESS.PROGRESS_DONE)
    THEN
      _eState                   := E_PROGRESS.PROGRESS_BUSY;
      _eRslt                    := _MoverItf[_nMover].Reset(FALSE);
    END_IF
END_CASE
//-----------------------------------------------------------------------------
//-----------------------------------------------------------------------------

MoverHaltAll                    := _eState;
END_METHOD

PROPERTY MoverInfo : REFERENCE TO ARRAY[1..MAX_MOVER] OF ST_MOVER_INFO
SET
_MoverInfo REF= MoverInfo;
END_SET
END_PROPERTY

PROPERTY MoverItf : reference TO ARRAY[1..MAX_MOVER] OF I_XtsTransport_Mover
SET
_MoverItf REF= MoverItf;
END_SET
END_PROPERTY

PROPERTY MoverLastGap : REFERENCE to ARRAY[1..MAX_MOVER] of LREAL
SET
_MoverLastGap REF= MoverLastGap;
END_SET
END_PROPERTY

PROPERTY MoverLastPosition : REFERENCE to ARRAY[1..MAX_MOVER] of LREAL
SET
_MoverLastPosition REF= MoverLastPosition;
END_SET
END_PROPERTY

METHOD MoverStopAll : e_progress
VAR_INPUT
  Execute     : BOOL;
END_VAR
VAR_INST
  _nMover     : UINT;
  _nErrorId   : UDINT;
  _eRslt,
  _eState     : E_PROGRESS;
  _stMoveData : ST_MOVE_DATA; // dyn constraints for _MoverItf[i].Halt(Execute, stMoveData)
END_VAR
//-----------------------------------------------------------------------------
IF NOT Execute 
THEN 
	_eState                       := E_PROGRESS.PROGRESS_INIT; 
END_IF 
//-----------------------------------------------------------------------------
IF NOT Check() 
THEN 
	MoverStopAll                  := E_PROGRESS.PROGRESS_ERROR; 
	RETURN; 
END_IF
//-----------------------------------------------------------------------------
//-----------------------------------------------------------------------------
CASE _eState
OF
  E_PROGRESS.PROGRESS_INIT:
    IF Execute
    THEN
      _nErrorId                 := 0;
      _nMover                   := 1;

      _eState                   := E_PROGRESS.PROGRESS_BUSY;

      IF (_eMessageLevel > E_MessageType.eMessageError)
      THEN
        _stMsg.eType            := E_MessageType.eMessageinfo;
        _stMsg.iErrorNumber     := 0;
        _stMsg.sText            := concat( 'State: ', TO_STRING(THIS^._eState));
        _stMsg.sText            := concat(_stMsg.sText, ': ');
        _stMsg.sText            := concat(_stMsg.sText, TO_STRING(_eState));
        f_MessageSet(_stMsg);
      END_IF
    END_IF
END_CASE
//-----------------------------------------------------------------------------
//-----------------------------------------------------------------------------
CASE _eState
OF
  E_PROGRESS.PROGRESS_BUSY:
    _eState                     := E_PROGRESS.PROGRESS_PREPARE;
    _stMoveData.rAcc            := _StationStart.rAccDec;
    _stMoveData.rGap            := _MoverLastGap[_nMover];

    _eRslt                      := _MoverItf[_nMover].Stop(FALSE, _stMoveData);
END_CASE
//-----------------------------------------------------------------------------
//-----------------------------------------------------------------------------
CASE _eState
OF
  E_PROGRESS.PROGRESS_PREPARE:
    _eRslt                      := _MoverItf[_nMover].Stop(TRUE, _stMoveData);

    IF (_eRslt = E_PROGRESS.PROGRESS_ERROR)
    THEN
      _eState                   := E_PROGRESS.PROGRESS_WORKING; // reset error on purpose, since we have to come back and get everybody in standstill
      _eRslt                    := _MoverItf[_nMover].Reset(FALSE);
      _nErrorId                 := _MoverInfo[_nMover].nErrorId; 

    ELSIF (_eRslt = E_PROGRESS.PROGRESS_DONE)
    THEN
      _eState                   := E_PROGRESS.PROGRESS_STARTUP;
    END_IF
END_CASE
//-----------------------------------------------------------------------------
//-----------------------------------------------------------------------------
CASE _eState
OF
  E_PROGRESS.PROGRESS_STARTUP:
    _eState                     := E_PROGRESS.PROGRESS_CHECK;
    _eRslt                      := _MoverItf[_nMover].Halt(FALSE, _stMoveData);
END_CASE
//-----------------------------------------------------------------------------
//-----------------------------------------------------------------------------
CASE _eState
OF
  E_PROGRESS.PROGRESS_CHECK:
    IF (_nMover > GVL_XTS.XpuInfo.nDetectedAxisCount-1)
    THEN
      _eState                   := E_PROGRESS.PROGRESS_OCCUPIED;
    ELSE
      _nMover                   := _nMover + 1;
      _eState                   := E_PROGRESS.PROGRESS_BUSY;
    END_IF
END_CASE
//-----------------------------------------------------------------------------
//-----------------------------------------------------------------------------
CASE _eState
OF
  E_PROGRESS.PROGRESS_OCCUPIED:
    IF (_GroupInfo.AllAxesStanding)
    THEN
      _eState                   := E_PROGRESS.PROGRESS_DONE;

      IF (_eMessageLevel > E_MessageType.eMessageError)
      THEN
        _stMsg.eType            := E_MessageType.eMessageInfo;
        _stMsg.eSubdevice       := e_Subdevice.TransportUnit_General;
        _stMsg.iErrorNumber     := 0;
        _stMsg.sText            := concat( 'State: ', TO_STRING(THIS^._eState));
        _stMsg.sText            := concat(_stMsg.sText, ': ');
        _stMsg.sText            := concat(_stMsg.sText, TO_STRING(_eState));
        f_MessageSet(_stMsg);
      END_IF
    ELSE
      _nMover                   := 1;
      _eState                   := E_PROGRESS.PROGRESS_BUSY;
    END_IF
END_CASE
//-----------------------------------------------------------------------------
//-----------------------------------------------------------------------------
CASE _eState
OF
  E_PROGRESS.PROGRESS_WORKING:
    _eRslt                      := _MoverItf[_nMover].Reset(TRUE);

    IF (_eRslt = E_PROGRESS.PROGRESS_ERROR)
    THEN
      _eRslt                    := _MoverItf[_nMover].Reset(FALSE);
      _nErrorId                 := _MoverInfo[_nMover].nErrorId; 

    ELSIF (_eRslt = E_PROGRESS.PROGRESS_DONE)
    THEN
      _eState                   := E_PROGRESS.PROGRESS_BUSY;
      _eRslt                    := _MoverItf[_nMover].Reset(FALSE);
    END_IF
END_CASE
//-----------------------------------------------------------------------------
//-----------------------------------------------------------------------------

MoverStopAll                    := _eState;
END_METHOD

PROPERTY State : REFERENCE TO ST_XTS_TRANSPORT_STATE
SET
_stState ref= State;
END_SET
END_PROPERTY

PROPERTY StationControl : REFERENCE TO ARRAY[1..MAX_STATION]  OF ST_STATION_CTRL
SET
_StationControl REF= StationControl;
END_SET
END_PROPERTY

PROPERTY StationCtrlItf : REFERENCE TO ARRAY[1..MAX_STATION]  OF I_XtsTransport_Station;
SET
_ItfStationCtrl REF= StationCtrlItf;
END_SET
END_PROPERTY

PROPERTY StationListsItf : reference to ARRAY[1..MAX_STATION] OF I_Station_LinkedList
SET
_ItfStationList ref= StationListsItf;
END_SET
END_PROPERTY

METHOD StationsClearAll : E_PROGRESS
VAR_INPUT
  Execute     : BOOL;
END_VAR
VAR_INST
  _nStation,
  _nErrorId   : UDINT;
  _eJobReslt,
  _eState     : E_PROGRESS;
END_VAR
//-----------------------------------------------------------------------------
IF NOT Execute 
THEN 
	_eState                       := E_PROGRESS.PROGRESS_INIT; 
END_IF 
//-----------------------------------------------------------------------------
IF NOT Check() 
THEN 
	StationsClearAll              := E_PROGRESS.PROGRESS_ERROR; 
	RETURN; 
END_IF
//-----------------------------------------------------------------------------
//-----------------------------------------------------------------------------
CASE _eState
OF
  E_PROGRESS.PROGRESS_INIT:
    IF Execute
    THEN
      _nErrorId                 := 0;
      _nStation                 := 1;
      _eState                   := E_PROGRESS.PROGRESS_BUSY;

      IF (_eMessageLevel > E_MessageType.eMessageError)
      THEN
        _stMsg.eType            := E_MessageType.eMessageInfo;
        _stMsg.iErrorNumber     := 0;
        _stMsg.sText            := concat( 'StationsClearAll: ', TO_STRING(THIS^._eState));
        _stMsg.sText            := concat(_stMsg.sText, ': ');
        _stMsg.sText            := concat(_stMsg.sText, TO_STRING(_eState));
        f_MessageSet(_stMsg);
      END_IF
    END_IF
  //---------------------------------------------------------------------------
  //---------------------------------------------------------------------------
  E_PROGRESS.PROGRESS_BUSY:
    // identity check, only valid stations are checked
    IF (_ItfStationCtrl[_nStation].StationId > 0)
    THEN
      _eState                   := E_PROGRESS.PROGRESS_PREPARE;

    ELSE
      _eState                   := E_PROGRESS.PROGRESS_WORKING;
    END_IF

  //---------------------------------------------------------------------------
  //---------------------------------------------------------------------------
  E_PROGRESS.PROGRESS_PREPARE:
    _eJobReslt                  := _ItfStationCtrl[_nStation].Init();

    IF (_eJobReslt = E_PROGRESS.PROGRESS_ERROR)
    THEN
      _eState                   := E_PROGRESS.PROGRESS_ERROR;
      _nErrorId                 := 669;

    ELSIF (_eJobReslt = E_PROGRESS.PROGRESS_DONE)
    THEN
      _eState                   := E_PROGRESS.PROGRESS_WORKING;
    END_IF

  //---------------------------------------------------------------------------
  //---------------------------------------------------------------------------
  E_PROGRESS.PROGRESS_WORKING:
    IF (_nStation < MAX_STATION)
    THEN
      _nStation                 := _nStation + 1;
      _eState                   := E_PROGRESS.PROGRESS_BUSY;
    ELSE
      _eState                   := E_PROGRESS.PROGRESS_DONE;

      IF (_eMessageLevel > E_MessageType.eMessageError)
      THEN
        _stMsg.eType            := E_MessageType.eMessageInfo;
        _stMsg.iErrorNumber     := 0;
        _stMsg.sText            := concat( 'StationsClearAll: ', TO_STRING(THIS^._eState));
        _stMsg.sText            := concat(_stMsg.sText, ': ');
        _stMsg.sText            := concat(_stMsg.sText, TO_STRING(_eState));
        f_MessageSet(_stMsg);
      END_IF
    END_IF
END_CASE
//-----------------------------------------------------------------------------
//-----------------------------------------------------------------------------

StationsClearAll                := _eState;
END_METHOD

METHOD StationsClearOutfeed : e_progress
VAR_INPUT
  Execute         : BOOL;
END_VAR
VAR_INST
  _StnState       : ST_STATION_STATE;

  _nStation,
  _nMover         : UINT;

  _nErrorId       : UDINT;

  _eRslt,
  _eState         : E_PROGRESS;
  
  _stMsg          : ST_Message;
  _stMoveData     : ST_MOVE_DATA;
END_VAR
//-----------------------------------------------------------------------------
IF NOT Execute 
THEN 
	_eState                       := E_PROGRESS.PROGRESS_INIT; 
END_IF 
//-----------------------------------------------------------------------------
IF NOT Check() 
THEN 
	StationsClearOutfeed           := E_PROGRESS.PROGRESS_ERROR; 
	RETURN; 
END_IF
//-----------------------------------------------------------------------------
//-----------------------------------------------------------------------------
CASE _eState
OF
  E_PROGRESS.PROGRESS_INIT:
    IF Execute
    THEN
      _nErrorId                 := 0;

      _nStation                 :=
      _nMover                   := 1;

      _eState                   := E_PROGRESS.PROGRESS_BUSY;

      IF (_eMessageLevel > E_MessageType.eMessageError)
      THEN
        _stMsg.eType            := E_MessageType.eMessageInfo;
        _stMsg.iErrorNumber     := 0;
        _stMsg.sText            := concat( 'StationsClearOutfeed: ', TO_STRING(THIS^._eState));
        _stMsg.sText            := concat(_stMsg.sText, ': ');
        _stMsg.sText            := concat(_stMsg.sText, TO_STRING(_eState));
        f_MessageSet(_stMsg);
      END_IF
    END_IF
END_CASE
//-----------------------------------------------------------------------------
//-----------------------------------------------------------------------------
CASE _eState
OF
  E_PROGRESS.PROGRESS_BUSY:
    _StnState                   := _StationState[_nStation];

    CASE _StnState.State
    OF
      E_STATION_STATE.STATION_MOVER_RELEASE,
      E_STATION_STATE.STATION_ERROR_OUTFEED_ERROR:
        _StationControl[_nStation].Cmd := E_STATION_CTRL.STATION_MOVER_GONE;

    ELSE
      _eState                   := E_PROGRESS.PROGRESS_PREPARE;  
    END_CASE
END_CASE
//-----------------------------------------------------------------------------
//-----------------------------------------------------------------------------
CASE _eState
OF
  E_PROGRESS.PROGRESS_PREPARE:
    IF (_nStation > MAX_STATION-1)
    THEN
      _eState                   := E_PROGRESS.PROGRESS_DONE;
    ELSE
      _nStation                 := _nStation + 1;
      _eState                   := E_PROGRESS.PROGRESS_BUSY;
    END_IF
END_CASE

StationsClearOutfeed             := _eState;
END_METHOD

PROPERTY StationStart : reference to ST_STATION_PARAMETER
SET
_StationStart REF= StationStart;
END_SET
END_PROPERTY

PROPERTY StationStartIndex : uint
GET
StationStartIndex := _nStartStation;
END_GET
SET
_nStartStation := StationStartIndex;
END_SET
END_PROPERTY

PROPERTY StationState : REFERENCE TO ARRAY[1..MAX_STATION]  OF ST_STATION_STATE
SET
_StationState REF= StationState;
END_SET
END_PROPERTY

METHOD Template : E_PROGRESS
VAR_INPUT
  Execute     : BOOL;
END_VAR
VAR_INST
  _nErrorId   : UDINT;
  _eState     : E_PROGRESS;
END_VAR
//-----------------------------------------------------------------------------
IF NOT Execute 
THEN 
	_eState                       := E_PROGRESS.PROGRESS_INIT; 
END_IF 
//-----------------------------------------------------------------------------
IF NOT Check() 
THEN 
	Template_1                    := E_PROGRESS.PROGRESS_ERROR; 
	RETURN; 
END_IF
//-----------------------------------------------------------------------------
//-----------------------------------------------------------------------------
CASE _eState
OF
  E_PROGRESS.PROGRESS_INIT:
    IF Execute
    THEN
      _nErrorId                 := 0;

      _eState                   := E_PROGRESS.PROGRESS_BUSY;
    END_IF
END_CASE
//-----------------------------------------------------------------------------
//-----------------------------------------------------------------------------
CASE _eState
OF
  E_PROGRESS.PROGRESS_BUSY:
    _eState                     := E_PROGRESS.PROGRESS_PREPARE;
END_CASE
//-----------------------------------------------------------------------------
//-----------------------------------------------------------------------------
CASE _eState
OF
  E_PROGRESS.PROGRESS_PREPARE:

    IF (.Error)
    THEN
      _eState                   := E_PROGRESS.PROGRESS_ERROR;
      _nErrorId                 := 


    ELSIF (.Done)
    THEN
      _eState                   := E_PROGRESS.;

    END_IF
END_CASE
//-----------------------------------------------------------------------------
//-----------------------------------------------------------------------------

Template_1                      := _eState;
END_METHOD

METHOD TransportRestart : e_progress // movers must already to be error free, enabled and added to CA Group
VAR_INPUT
  Execute         : BOOL;
END_VAR
VAR_INST
  _StnState       : ST_STATION_STATE;

  _nStation,
  _nMover         : UINT;

  _nErrorId       : UDINT;

  _eRslt,
  _eState         : E_PROGRESS;
  
  _stMsg          : ST_Message;
  _stMoveData     : ST_MOVE_DATA;
END_VAR
//-----------------------------------------------------------------------------
IF NOT Execute 
THEN 
	_eState                       := E_PROGRESS.PROGRESS_INIT; 
END_IF 
//-----------------------------------------------------------------------------
IF NOT Check() 
THEN 
	TransportRestart              := E_PROGRESS.PROGRESS_ERROR; 
	RETURN; 
END_IF
//-----------------------------------------------------------------------------
//-----------------------------------------------------------------------------
CASE _eState
OF
  E_PROGRESS.PROGRESS_INIT:
    IF Execute
    THEN
      _nErrorId                 := 0;

      _nStation                 :=
      _nMover                   := 1;

      IF (_GroupInfo.AxisCountEnabled = GVL_XTS.XpuInfo.nDetectedAxisCount)
      THEN
        _eState                 := E_PROGRESS.PROGRESS_BUSY;

        IF (_eMessageLevel > E_MessageType.eMessageError)
        THEN
          _stMsg.eType          := E_MessageType.eMessageinfo;
          _stMsg.eSubdevice     := e_Subdevice.TransportUnit_Restart;
          _stMsg.iErrorNumber   := 0;
          _stMsg.sText          := concat( 'State: ', TO_STRING(THIS^._eState));
          _stMsg.sText          := concat(_stMsg.sText, ': ');
          _stMsg.sText          := concat(_stMsg.sText, TO_STRING(_eState));
          f_MessageSet(_stMsg);
        END_IF
      ELSE
        _eState                 := E_PROGRESS.PROGRESS_ERROR;

        _stMsg.eType            := E_MessageType.eMessageError;
        _stMsg.eSubdevice       := e_Subdevice.TransportUnit_Restart;
        _stMsg.iErrorNumber     := _GroupInfo.AxisCountEnabled;
        _stMsg.sText            := TO_STRING(_eState);
        _stMsg.sText            := concat(_stMsg.sText, ': _GroupInfo.AxisCountEnabled <> GVL_XTS.XpuInfo.nDetectedAxisCount');
        f_MessageSet(_stMsg);
      END_IF
    END_IF
END_CASE
//-----------------------------------------------------------------------------
//-----------------------------------------------------------------------------
CASE _eState
OF
  E_PROGRESS.PROGRESS_BUSY:
    _StnState                   := _StationState[_nStation];

    CASE _StnState.State
    OF
      E_STATION_STATE.STATION_ERROR_INFEED_ERROR:
        _StationControl[_nStation].Cmd := E_STATION_CTRL.STATION_MOVER_ENTER_RETRY;

      E_STATION_STATE.STATION_MOVER_RELEASE,
      E_STATION_STATE.STATION_ERROR_OUTFEED_ERROR:
        _StationControl[_nStation].Cmd := E_STATION_CTRL.STATION_MOVER_GONE;

      E_STATION_STATE.STATION_ERROR_FATAL:
        _eState                 := E_PROGRESS.PROGRESS_ERROR;

        _stMsg.eType            := E_MessageType.eMessageError;
        _stMsg.eSubdevice       := e_Subdevice.TransportUnit_Restart;
        _stMsg.iErrorNumber     := _nStation;
        _stMsg.sText            := TO_STRING(_eState);
        _stMsg.sText            := concat(_stMsg.sText, ': _nStation STATION_ERROR_FATAL');
        f_MessageSet(_stMsg);

    ELSE
      _eState                   := E_PROGRESS.PROGRESS_PREPARE;  
    END_CASE
END_CASE
//-----------------------------------------------------------------------------
//-----------------------------------------------------------------------------
CASE _eState
OF
  E_PROGRESS.PROGRESS_PREPARE:
    IF (_nStation > MAX_STATION-1)
    THEN
      _eState                   := E_PROGRESS.PROGRESS_STARTUP;
    ELSE
      _nStation                 := _nStation + 1;
      _eState                   := E_PROGRESS.PROGRESS_BUSY;
    END_IF
END_CASE
//-----------------------------------------------------------------------------
//-----------------------------------------------------------------------------
CASE _eState
OF
  E_PROGRESS.PROGRESS_STARTUP:
    _stMoveData.rPos            := _MoverLastPosition[_nMover];
    _stMoveData.rGap            := _MoverLastGap     [_nMover];

    _stMoveData.rVelo           := _StationStart.rVelo;
    _stMoveData.rAcc            := _StationStart.rAccDec;
    _stMoveData.rJerk           := _StationStart.rJerk;

    _stMoveData.rDelta          :=   0.1;
    _stMoveData.rDistance       :=  -1.0;
    _stMoveData.rOverride       := 100.0;

    _eRslt                      := _MoverItf[_nMover].SendToAbsPosCa(FALSE, _stMoveData);

    IF (_MoverInfo[_nMover].bMoverEnabled)
    THEN
      _eState                   := E_PROGRESS.PROGRESS_CHECK;
    END_IF
END_CASE
//-----------------------------------------------------------------------------
//-----------------------------------------------------------------------------
CASE _eState
OF
  E_PROGRESS.PROGRESS_CHECK:
    _eRslt                      := _MoverItf[_nMover].SendToAbsPosCa(TRUE, _stMoveData);

    IF (_eRslt = E_PROGRESS.PROGRESS_ERROR)
    THEN
      _eState                   := E_PROGRESS.PROGRESS_ERROR;

    ELSIF (_eRslt = E_PROGRESS.PROGRESS_DONE)
    THEN
      _eRslt                    := _MoverItf[_nMover].SendToAbsPosCa(FALSE, _stMoveData);
      _eState                   := E_PROGRESS.PROGRESS_OCCUPIED;
    END_IF
END_CASE
//-----------------------------------------------------------------------------
//-----------------------------------------------------------------------------
CASE _eState
OF
  E_PROGRESS.PROGRESS_OCCUPIED:
    IF (_nMover > GVL_XTS.XpuInfo.nDetectedAxisCount-1)
    THEN
      _eState                   := E_PROGRESS.PROGRESS_DONE;

      IF (_eMessageLevel > E_MessageType.eMessageError)
      THEN
        _stMsg.eType            := E_MessageType.eMessageInfo;
        _stMsg.eSubdevice       := e_Subdevice.TransportUnit_General;
        _stMsg.iErrorNumber     := 0;
        _stMsg.sText            := concat( 'State: ', TO_STRING(THIS^._eState));
        _stMsg.sText            := concat(_stMsg.sText, ': ');
        _stMsg.sText            := concat(_stMsg.sText, TO_STRING(_eState));
        f_MessageSet(_stMsg);
      END_IF
      GVL_MSG_XTS.TransportMessageCtrl.Cmd  := E_MESSAGE_CTRL.MSG_CTRL_WRITE;
    ELSE
      _nMover                   := _nMover + 1;
      _eState                   := E_PROGRESS.PROGRESS_STARTUP;
    END_IF
END_CASE
//-----------------------------------------------------------------------------
//-----------------------------------------------------------------------------

TransportRestart                := _eState;
END_METHOD

METHOD TransportStart : e_progress
VAR_INPUT
  Execute       : BOOL;
END_VAR
VAR_INST
  _nMover,
  _nStation     : UINT;
  _nErrorId     : UDINT;

  _stMoveData   : ST_MOVE_DATA;

  _eRslt,
  _eStateError,
  _eState       : E_PROGRESS;
END_VAR
//-----------------------------------------------------------------------------
IF NOT Execute 
THEN 
	_eState                       := E_PROGRESS.PROGRESS_INIT; 
END_IF 
//-----------------------------------------------------------------------------
IF NOT Check() 
THEN 
	TransportStart                := E_PROGRESS.PROGRESS_ERROR; 
	RETURN; 
END_IF
//-----------------------------------------------------------------------------
//-----------------------------------------------------------------------------
CASE _eState
OF
  E_PROGRESS.PROGRESS_INIT:
    IF Execute
    THEN
      _nErrorId                 := 0;
      _nMover                   := 1;

      IF (_StationStart.rPosWait - (_MoverInfo[_nMover].rModuloActPos +0.1) < 0)
      THEN
        _stMoveData.rPos        := _StationStart.rPosWait + _MoverItf[_nMover].RailLength;
      ELSE
        _stMoveData.rPos        := _StationStart.rPosWait;
      END_IF

      _stMoveData.rGap          := _StationStart.rGap;

      _stMoveData.rVelo         := _StationStart.rVelo;
      _stMoveData.rAcc          := _StationStart.rAccDec;
      _stMoveData.rJerk         := _StationStart.rJerk;

      _stMoveData.rDelta        :=   0.05;
      _stMoveData.rDistance     :=  -1.0;     // distance used by SendToPosCa

      _stMoveData.rOverride     := 100.0;

      _eRslt                    := _MoverItf[_nMover].SendToModuloPosCa(FALSE, _stMoveData);
      _eRslt                    := _MoverItf[_nMover].SendToAbsPosCa(FALSE, _stMoveData);
      _eRslt                    := StationsClearAll(FALSE);

      IF (_GroupInfo.AxisCountEnabled = _XpuInfo.nDetectedAxisCount) AND
         (_XpuInfo.nDetectedAxisCount > 0)
      THEN
        _eState                 := E_PROGRESS.PROGRESS_BUSY;

        IF (_eMessageLevel > E_MessageType.eMessageError)
        THEN
          _stMsg.eType          := E_MessageType.eMessageinfo;
          _stMsg.eSubdevice     := e_Subdevice.TransportUnit_Start;
          _stMsg.iErrorNumber   := 0;
          _stMsg.sText          := concat( 'State: ', TO_STRING(THIS^._eState));
          _stMsg.sText          := concat(_stMsg.sText, ': ');
          _stMsg.sText          := concat(_stMsg.sText, TO_STRING(_eState));
          f_MessageSet(_stMsg);
        END_IF
      ELSE
        _eStateError            := _eState;
        _eState                 := E_PROGRESS.PROGRESS_ERROR;

        _stMsg.eType            := E_MessageType.eMessageError;
        _stMsg.eSubdevice       := e_Subdevice.TransportUnit_Start;
        _stMsg.iErrorNumber     := _GroupInfo.AxisCountEnabled;
        _stMsg.sText            := TO_STRING(_eState);
        _stMsg.sText            := concat(_stMsg.sText, ': _GroupInfo.AxisCountEnabled <> MAX_MOVER');
        f_MessageSet(_stMsg);
      END_IF
    END_IF

  //---------------------------------------------------------------------------
  E_PROGRESS.PROGRESS_BUSY:
    _eRslt                      := StationsClearAll(TRUE); // all xts station queues clear
    IF (_eRslt = E_PROGRESS.PROGRESS_DONE)
    THEN
      _eState                   := E_PROGRESS.PROGRESS_PREPARE;
    ELSE
      IF (_eRslt = E_PROGRESS.PROGRESS_ERROR)
      THEN
        _eStateError            := _eState;
        _eState                 := E_PROGRESS.PROGRESS_ERROR;
      END_IF
    END_IF

  E_PROGRESS.PROGRESS_PREPARE:
    _eRslt                      := _MoverItf[_nMover].SendToModuloPosCa(TRUE, _stMoveData);

    IF (_eRslt = E_PROGRESS.PROGRESS_ERROR)
    THEN
      _eStateError              := _eState;
      _eState                   := E_PROGRESS.PROGRESS_ERROR;
      _nErrorId                 := _MoverInfo[_nMover].nErrorId;
      _eRslt                    := _MoverItf[_nMover].SendToModuloPosCa(FALSE, _stMoveData); 

    ELSIF (_eRslt = E_PROGRESS.PROGRESS_DONE)
    THEN
      _eState                   := E_PROGRESS.PROGRESS_STARTUP;
      _eRslt                    := _MoverItf[_nMover].SendToModuloPosCa(FALSE, _stMoveData);
    END_IF

  //---------------------------------------------------------------------------
  E_PROGRESS.PROGRESS_STARTUP:
    IF (_nMover > GVL_XTS.XpuInfo.nDetectedAxisCount-1)
    THEN
      // all mover are sent to start position, now prepare ticket for Mover 1
      _eState                         := E_PROGRESS.PROGRESS_CHECK;
      // ticket data
      _stMoverDataSend.nMask          := TO_USINT(EXPT(2,_StationStart.nConfiguredStopCount))-1;
      _stMoverDataSend.nMoverId       := TO_USINT(1);
      _stMoverDataSend.nTargetStation := TO_USINT(_nStartStation);
  
      IF (_nStartStation > 0) AND
         (_nStartStation < MAX_STATION+1)
      THEN
        _stListResult           := _ItfStationList[_nStartStation].AddTailValue(_stMoverDataSend); // add first mover to list of _ItfStations[_nStartStation]
      END_IF

    ELSE
      _nMover                   := _nMover + 1;                                                 // increment mover ID
      _stMoveData.rPos          := _StationStart.rPosWait + 2*_MoverItf[_nMover].RailLength;    // all other mover are commanded an extra round, to make sure that mover 1 is always leading the pack
      _eRslt                    := _MoverItf[_nMover].SendToModuloPosCa(FALSE, _stMoveData);
      _eRslt                    := _MoverItf[_nMover].SendToAbsPosCa(FALSE, _stMoveData);
      _eState                   := E_PROGRESS.PROGRESS_PREPARE;                                 // go back and trigger move
    END_IF

  //---------------------------------------------------------------------------
  E_PROGRESS.PROGRESS_CHECK:
    IF (_MoverInfo[1].bMoverInTarget)
    THEN
      IF (_GroupInfo.AllAxesStanding) // wait for all mover standstill
      THEN
        _stMoveData.rPos        := _MoverInfo[1].rAbsTargetPos;                    // Mover1 position to retrigger the movers

        IF (MAX_MOVER > 1)
        THEN
          _nMover               := 2;
          IF (_stMoveData.rPos < _MoverInfo[_nMover].rAbsActPos)
          THEN
            _stMoveData.rPos    := _stMoveData.rPos + _MoverItf[_nMover].RailLength;
          END_IF
          _eState               := E_PROGRESS.PROGRESS_OCCUPIED;
        ELSE
          _eState               := E_PROGRESS.PROGRESS_WORKING;
        END_IF
      END_IF
    END_IF

  //---------------------------------------------------------------------------
  E_PROGRESS.PROGRESS_OCCUPIED:
    _eRslt                      := _MoverItf[_nMover].SendToAbsPosCa(TRUE, _stMoveData); // retrigger

    IF (_eRslt = E_PROGRESS.PROGRESS_ERROR)
    THEN
      _eStateError              := _eState;
      _eState                   := E_PROGRESS.PROGRESS_ERROR;
      _nErrorId                 := _MoverInfo[_nMover].nErrorId;
      _eRslt                    := _MoverItf[_nMover].SendToAbsPosCa(FALSE, _stMoveData); 

    ELSIF (_eRslt = E_PROGRESS.PROGRESS_DONE)
    THEN
      _eState                   := E_PROGRESS.PROGRESS_WORKING;
      _eRslt                    := _MoverItf[_nMover].SendToAbsPosCa(FALSE, _stMoveData);

      // write ticket for mover in station list
      _stMoverDataSend.nMask          := TO_USINT(EXPT(2,_StationStart.nConfiguredStopCount))-1;
      _stMoverDataSend.nMoverId       := TO_USINT(_nMover);
      _stMoverDataSend.nTargetStation := TO_USINT(_nStartStation);

      IF (_nStartStation > 0) AND
         (_nStartStation < MAX_STATION+1)
      THEN
        _stListResult                 := _ItfStationList[_nStartStation].AddTailValue(_stMoverDataSend); // enter in list
      END_IF
    END_IF

  //---------------------------------------------------------------------------
  E_PROGRESS.PROGRESS_WORKING:
    IF (_nMover > GVL_XTS.XpuInfo.nDetectedAxisCount-1)
    THEN
      _eState                   := E_PROGRESS.PROGRESS_DONE;

      IF (_eMessageLevel > E_MessageType.eMessageError)
      THEN
        _stMsg.eType            := E_MessageType.eMessageInfo;
        _stMsg.eSubdevice       := e_Subdevice.TransportUnit_Start;
        _stMsg.iErrorNumber     := 0;
        _stMsg.sText            := concat( 'State: ', TO_STRING(THIS^._eState));
        _stMsg.sText            := concat(_stMsg.sText, ': ');
        _stMsg.sText            := concat(_stMsg.sText, TO_STRING(_eState));
        f_MessageSet(_stMsg);
      END_IF
      GVL_MSG_XTS.TransportMessageCtrl.Cmd  := E_MESSAGE_CTRL.MSG_CTRL_WRITE;
    ELSE
      _nMover                   := _nMover + 1;
      IF (_stMoveData.rPos < _MoverInfo[_nMover].rAbsActPos)
      THEN
        _stMoveData.rPos        := _stMoveData.rPos + _MoverItf[_nMover].RailLength;
      END_IF
      _eState                   := E_PROGRESS.PROGRESS_OCCUPIED;
    END_IF
END_CASE
//-----------------------------------------------------------------------------
//-----------------------------------------------------------------------------

TransportStart                  := _eState;
END_METHOD

PROPERTY XpuCtrl : REFERENCE TO ST_XPU_CTRL
SET
_XpuCtrl REF= XpuCtrl;
END_SET
END_PROPERTY

PROPERTY XpuInfo : REFERENCE TO ST_XPU_INFO
SET
_XpuInfo REF= XpuInfo;
END_SET
END_PROPERTY

METHOD XpuInit : E_PROGRESS
VAR_INPUT
  Execute     : BOOL;
END_VAR
VAR_INST
  _nErrorId   : UDINT;
  _eJobReslt,
  _eState     : E_PROGRESS;
END_VAR
//-----------------------------------------------------------------------------
IF NOT Execute 
THEN 
	_eState                       := E_PROGRESS.PROGRESS_INIT; 
END_IF 
//-----------------------------------------------------------------------------
IF NOT Check() 
THEN 
	XpuInit                       := E_PROGRESS.PROGRESS_ERROR; 
	RETURN; 
END_IF
//-----------------------------------------------------------------------------
//-----------------------------------------------------------------------------
CASE _eState
OF
  E_PROGRESS.PROGRESS_INIT:
    IF Execute
    THEN
      _nErrorId                 := 0;
      _XpuCtrl.Cmd              := E_XPU_CTRL.XTS_CMD_NULL; // clear interface

      _eState                   := E_PROGRESS.PROGRESS_BUSY;
    END_IF
  //---------------------------------------------------------------------------
  //---------------------------------------------------------------------------
  E_PROGRESS.PROGRESS_BUSY:
    _XpuCtrl.Cmd                := E_XPU_CTRL.XTS_CMD_INIT; // start Xpu init

    IF (f_GetProgress(_XpuState.State) = E_PROGRESS.PROGRESS_DONE)         // check Xpu init done
    THEN
      _eState                   := E_PROGRESS.PROGRESS_PREPARE;

    ELSIF (f_GetProgress(_XpuState.State) = E_PROGRESS.PROGRESS_ERROR)     // check for error
    THEN
      _eState                   := E_PROGRESS.PROGRESS_ERROR;
    END_IF
  //---------------------------------------------------------------------------
  //---------------------------------------------------------------------------
  E_PROGRESS.PROGRESS_PREPARE:
    _XpuCtrl.Cmd                := E_XPU_CTRL.XTS_IDLE;     // Xpu start cyclic checks and mover detection

    IF (f_GetProgress(_XpuState.State) = E_PROGRESS.PROGRESS_ERROR)     // check for error
    THEN
      _eState                   := E_PROGRESS.PROGRESS_ERROR;

    ELSIF (f_GetProgress(_XpuState.State) = E_PROGRESS.PROGRESS_WORKING)      // check Xpu Idle working
    THEN
      _eState                   := E_PROGRESS.PROGRESS_STARTUP;

    END_IF
  //---------------------------------------------------------------------------
  //---------------------------------------------------------------------------
  E_PROGRESS.PROGRESS_STARTUP:
    IF (f_GetProgress(_XpuState.State) = E_PROGRESS.PROGRESS_ERROR)
    THEN
      _eState                   := E_PROGRESS.PROGRESS_ERROR;

    ELSIF (_XpuState.Check = E_XPU_CHECK.MOVER_ID_SIMULATION) OR
          (_XpuState.Check = E_XPU_CHECK.MOVER_ID_STANDARD)   OR
          (_XpuState.Check = E_XPU_CHECK.MOVER_ID_DETECTION_VALID)
    THEN
      _eState                   := E_PROGRESS.PROGRESS_DONE;

      IF (_eMessageLevel = E_MessageType.eMessageVerbose)
      THEN
        _stMsg.eType            := E_MessageType.eMessageVerbose;
        _stMsg.eSubdevice       := e_Subdevice.TransportUnit_General;
        _stMsg.iErrorNumber     := 0;
        _stMsg.sText            := concat( 'State: ', TO_STRING(THIS^._eState));
        _stMsg.sText            := concat(_stMsg.sText, ': ');
        _stMsg.sText            := concat(_stMsg.sText, TO_STRING(_eState));
        f_MessageSet(_stMsg);
      END_IF
    END_IF
END_CASE
//-----------------------------------------------------------------------------
//-----------------------------------------------------------------------------
XpuInit                         := _eState;
END_METHOD

PROPERTY XpuState : REFERENCE TO ST_XPU_STATE
SET
_XpuState ref= XpuState;
END_SET
END_PROPERTY

END_FUNCTION_BLOCK

(* stored: Version 1.1.0.1, ProductVersion 3.1.4026.18
   POU fb_TransportUnit: Id {0ce87c95-a3e8-4212-b1c2-ee9df67705ee}, SpecialFunc None
   Folder methods: Id {0fe230de-36ae-4b97-83bc-6faccc9a05f7}
   Folder private: Id {79e5ca92-d9a5-425b-90ee-09934802d3c9}
   Folder properties: Id {79f5ed1f-7f7f-465b-8c47-d008b4dc44a2}
   Method Check: Id {cf27f3cc-50a5-4b1d-800c-93c52928c8a9}
   Method Cmd: Id {30bf2167-af11-4fc4-9325-16711ff925c6}
   Property Ctrl: Id {bf641ce2-0f39-4e29-b10a-7cd092476a93}
   Set Set: Id {87c918b6-6dc5-4a7a-8522-32056df06ad1}
   Method GroupBuild: Id {6560d614-3027-47d4-ab3b-0c99f0adeee0}
   Method GroupClear: Id {02b20a3a-d2af-452a-8e64-30135bd02948}
   Method GroupEnable: Id {bd2aede9-73ce-449c-97e3-f8856b827d01}
   Property GroupInfo: Id {eb8b9079-c486-4292-ab0d-e91edc853d54}
   Set Set: Id {28279787-7f62-474a-83c3-b06bfc4033b6}
   Property GroupItf: Id {5830bcb9-927c-4649-bfa5-dc6af0c4ef87}
   Set Set: Id {0836a44a-6504-4efb-ad0f-8cf37108710f}
   Method GroupStop: Id {0d086cb6-c6e5-48dd-8ec6-2cdceaa79a8e}
   Property MessageLevel: Id {cd92ca61-0c87-402d-9e64-d40bf3904b0a}
   Set Set: Id {3fc519db-7a0d-413d-8895-e7e2a525ad76}
   Method MoverDisableAll: Id {dfd3e28f-9149-411c-a9a0-e7fbedcee60a}
   Method MoverEnableAll: Id {c143a5c1-7d6a-4782-ad06-eb72e3e7b1e3}
   Method MoverHaltAll: Id {cc2e5e06-12c3-46fb-b8b0-3014c6d7dab4}
   Property MoverInfo: Id {efe23682-e809-4361-a57c-83cc4839891a}
   Set Set: Id {4804ae7c-4ea6-4aef-9370-3fc423ea6ed9}
   Property MoverItf: Id {c0185cf8-8f4e-47ad-9854-5b38a7c29416}
   Set Set: Id {e2836124-e67f-4103-a0d4-754562413f76}
   Property MoverLastGap: Id {12d22cab-bad7-41fc-9d68-adc96ec322fe}
   Set Set: Id {fa5acb95-48a8-4795-a0ab-fef5428ca8dc}
   Property MoverLastPosition: Id {2be09d03-f746-4871-ba7e-12bb061a6a9c}
   Set Set: Id {fcd11e7d-3d01-4d4f-98b0-98a6ff9632a0}
   Method MoverStopAll: Id {3d55d9ea-f977-4be0-bc91-dfb146bd2bbb}
   Property State: Id {1debc73a-7f5c-41d2-b68f-665e692b5c49}
   Set Set: Id {0cba4462-93ee-4d88-8c2e-c534aa587382}
   Property StationControl: Id {eb73d392-fdf8-4999-8a70-4f14a0de048a}
   Set Set: Id {48c36e60-58ac-40d7-99d4-1897012350e2}
   Property StationCtrlItf: Id {ba5c1e1d-dd07-4ce3-b818-96dfcfc382e7}
   Set Set: Id {ca882bea-1de3-4552-8d14-c5726862d2df}
   Property StationListsItf: Id {c1a5b764-3f6c-49d5-bb0c-3b39c0690736}
   Set Set: Id {0952c75c-3bbc-4b64-8624-7e4b6e37cd53}
   Method StationsClearAll: Id {da099dc4-d96b-43fb-b7bd-5b5d7c7104e0}
   Method StationsClearOutfeed: Id {5a55f4b0-2e71-4a29-bbda-ee132d22fc6c}
   Property StationStart: Id {9e259b8c-8238-454a-ae35-ccd1cef99baf}
   Set Set: Id {792867b6-c5c6-4624-8f17-698b7d9294c0}
   Property StationStartIndex: Id {84465866-3566-443c-8dc8-a47caea54b63}
   Get Get: Id {969c1fda-0f45-4fa1-badd-49dfab8aa29a}
   Set Set: Id {4f0a04d5-ea72-4804-9524-32751df5066b}
   Property StationState: Id {952bfdaf-ee8f-4a1f-8fd3-050f5e1c84d8}
   Set Set: Id {c4f6b766-cd17-4e88-b784-22a9e492ccb2}
   Method Template: Id {0aa0dd39-83ae-40d2-a365-a70ee97877b0}
   Method TransportRestart: Id {b5813896-5bda-4193-aba0-c07a9ac4ce2c}
   Method TransportStart: Id {cc22b853-18d6-4249-9a4d-acf2fc6c4a7c}
   Property XpuCtrl: Id {d96d119e-1863-494a-8419-7489c5dd721e}
   Set Set: Id {b2dc03c5-15d5-441f-b3fb-4200f2a1805b}
   Property XpuInfo: Id {67f137b2-091c-400c-ad52-7d4612b91604}
   Set Set: Id {ddf59d08-eae4-4c75-8899-fb5e74a616f7}
   Method XpuInit: Id {5e389358-507c-4c35-9d4a-3ac76b3c0d17}
   Property XpuState: Id {d619b5da-22c5-4ef3-b5fa-6142e558f71a}
   Set Set: Id {70f24a57-e57a-48dc-be92-700e52e5fd17} *)
